TYPE E_Command :
(
	None,
	Start,
	Stop,
	Reset
);
END_TYPE

(* stored: Version 1.1.0.1, ProductVersion 3.1.4024.12
   DUT E_Command: Id {6d412786-217f-43c2-bcc4-af5c3e616d71} *)
